// TIA Portal V18 export
TYPE "LGasp_Monitoraggi"
// stored: IsFailsafeCompliant false
   STRUCT
      nome : String := '-';
      abilitato : Bool;
      intervenuto : Bool;
      reset : Bool;
   END_STRUCT;
END_TYPE
